# EPICS autosave request: mcaApp/Db/icb_amp_settings.req
# FILE... icb_amp_settings.req
# USAGE.. icb_amp.db fields autosave'd.
$(P)$(AMP)CGAIN
$(P)$(AMP)FGAIN
$(P)$(AMP)SFGAIN
$(P)$(AMP)INPP
$(P)$(AMP)INHP
$(P)$(AMP)DMOD
$(P)$(AMP)SMOD
$(P)$(AMP)PTYP
$(P)$(AMP)PURMOD
$(P)$(AMP)BLMOD
$(P)$(AMP)DTMOD
$(P)$(AMP)PZ
